PROGRAM GL5B_Accumulation
VAR
	
	RUN_FWD_TO_GL2_BIT : BOOL; // GL2 EMPTY SO SEND PART FROM GL5B TO GL2
	RUN_FWD_TO_EXIT_BIT : BOOL; // RUN GL5B FWD TO EXIT SENSOR
	
END_VAR
VAR // added by the converter: edge detectors and wires of the graphical bodies
    _w1 : BOOL;
END_VAR

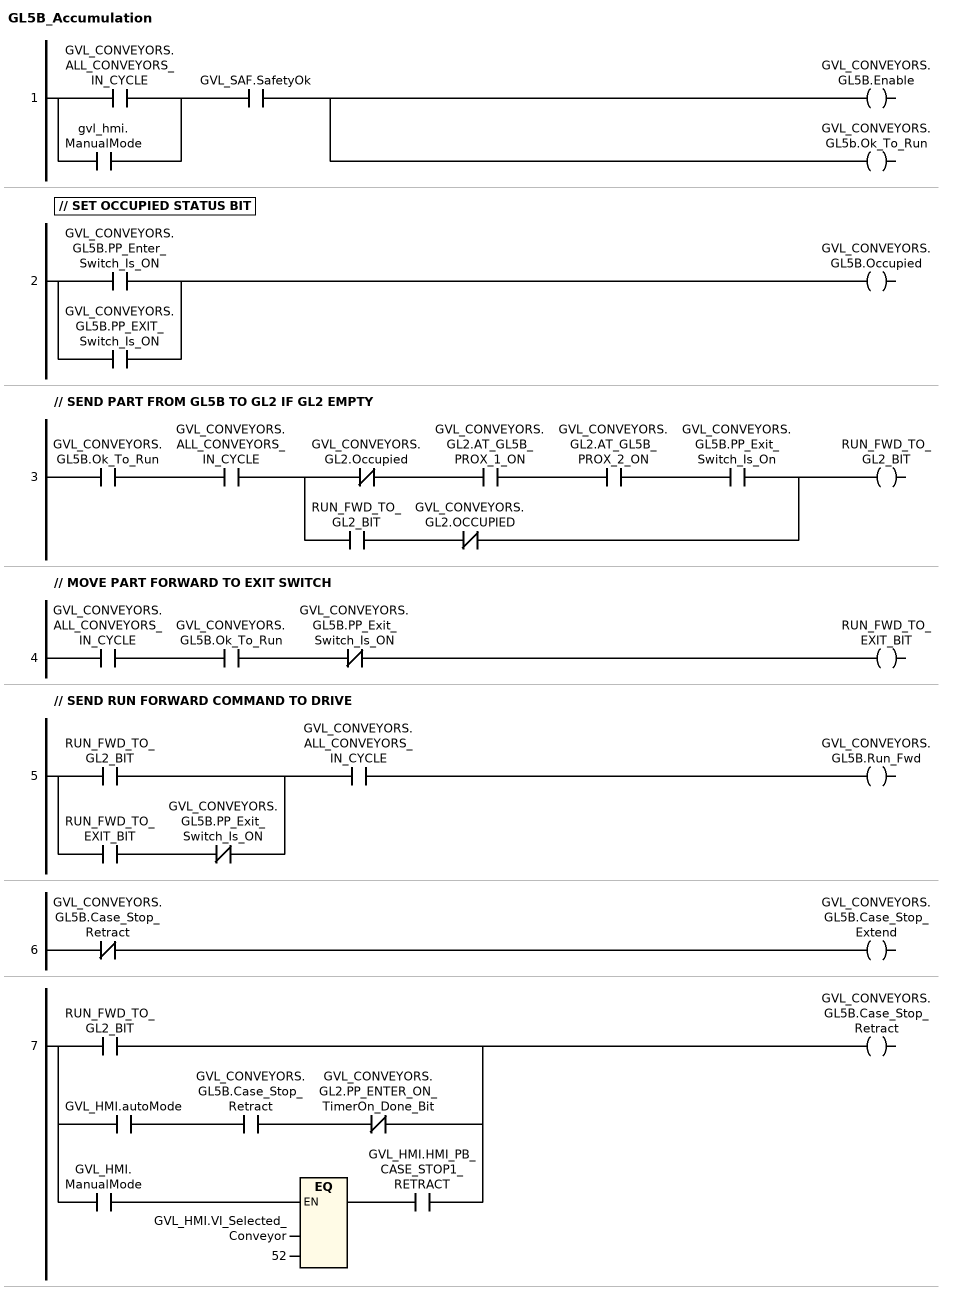
// NETWORK 1
_w1 := (GVL_CONVEYORS.ALL_CONVEYORS_IN_CYCLE OR gvl_hmi.ManualMode) AND GVL_SAF.SafetyOk;
GVL_CONVEYORS.GL5B.Enable := _w1;
GVL_CONVEYORS.GL5b.Ok_To_Run := _w1;

// NETWORK 2
// label: // SET OCCUPIED STATUS BIT
GVL_CONVEYORS.GL5B.Occupied := GVL_CONVEYORS.GL5B.PP_Enter_Switch_Is_ON OR GVL_CONVEYORS.GL5B.PP_EXIT_Switch_Is_ON;

// NETWORK 3: // SEND PART FROM GL5B TO GL2 IF GL2 EMPTY
RUN_FWD_TO_GL2_BIT := GVL_CONVEYORS.GL5B.Ok_To_Run AND GVL_CONVEYORS.ALL_CONVEYORS_IN_CYCLE AND (NOT GVL_CONVEYORS.GL2.Occupied AND GVL_CONVEYORS.GL2.AT_GL5B_PROX_1_ON AND GVL_CONVEYORS.GL2.AT_GL5B_PROX_2_ON AND GVL_CONVEYORS.GL5B.PP_Exit_Switch_Is_On OR RUN_FWD_TO_GL2_BIT AND NOT GVL_CONVEYORS.GL2.OCCUPIED);

// NETWORK 4: // MOVE PART FORWARD TO EXIT SWITCH
RUN_FWD_TO_EXIT_BIT := GVL_CONVEYORS.ALL_CONVEYORS_IN_CYCLE AND GVL_CONVEYORS.GL5B.Ok_To_Run AND NOT GVL_CONVEYORS.GL5B.PP_Exit_Switch_Is_ON;

// NETWORK 5: // SEND RUN FORWARD COMMAND TO DRIVE
GVL_CONVEYORS.GL5B.Run_Fwd := (RUN_FWD_TO_GL2_BIT OR RUN_FWD_TO_EXIT_BIT AND NOT GVL_CONVEYORS.GL5B.PP_Exit_Switch_Is_ON) AND GVL_CONVEYORS.ALL_CONVEYORS_IN_CYCLE;

// NETWORK 6
GVL_CONVEYORS.GL5B.Case_Stop_Extend := NOT GVL_CONVEYORS.GL5B.Case_Stop_Retract;

// NETWORK 7
GVL_CONVEYORS.GL5B.Case_Stop_Retract := RUN_FWD_TO_GL2_BIT OR GVL_HMI.autoMode AND GVL_CONVEYORS.GL5B.Case_Stop_Retract AND NOT GVL_CONVEYORS.GL2.PP_ENTER_ON_TimerOn_Done_Bit OR (GVL_HMI.ManualMode AND GVL_HMI.VI_Selected_Conveyor = 52) AND GVL_HMI.HMI_PB_CASE_STOP1_RETRACT;

END_PROGRAM

(* stored: Version 1.1.0.1, ProductVersion 3.1.4024.12
   POU GL5B_Accumulation: Id {ae7e7637-c93c-4317-a23b-6db03add0692}, SpecialFunc None *)
